// TIA Portal V20 export
DATA_BLOCK "DB_AsiSetpoint"   // DB31
// stored: Access Published, MemoryReserve 100, Namespace LineA1
   VAR
      Line : Struct
         A1 : Struct
            DirChange : Struct
               Conveyor : Array[_.minA1.._.maxA1] of Bool;
            END_STRUCT;
            Speed : Struct
               Conveyor : Array[_.minA1.._.maxA1] of Bool;
            END_STRUCT;
         END_STRUCT;
      END_STRUCT;
   END_VAR
BEGIN
   // Line.A1.DirChange.Conveyor[1001] : AS1.1.1
   // Line.A1.DirChange.Conveyor[1002] : AS1.1.2
   // Line.A1.Speed.Conveyor[1001] : AS1.1.1
   // Line.A1.Speed.Conveyor[1002] : AS1.1.2
END_DATA_BLOCK
